RoboDK station: ex2.rdk

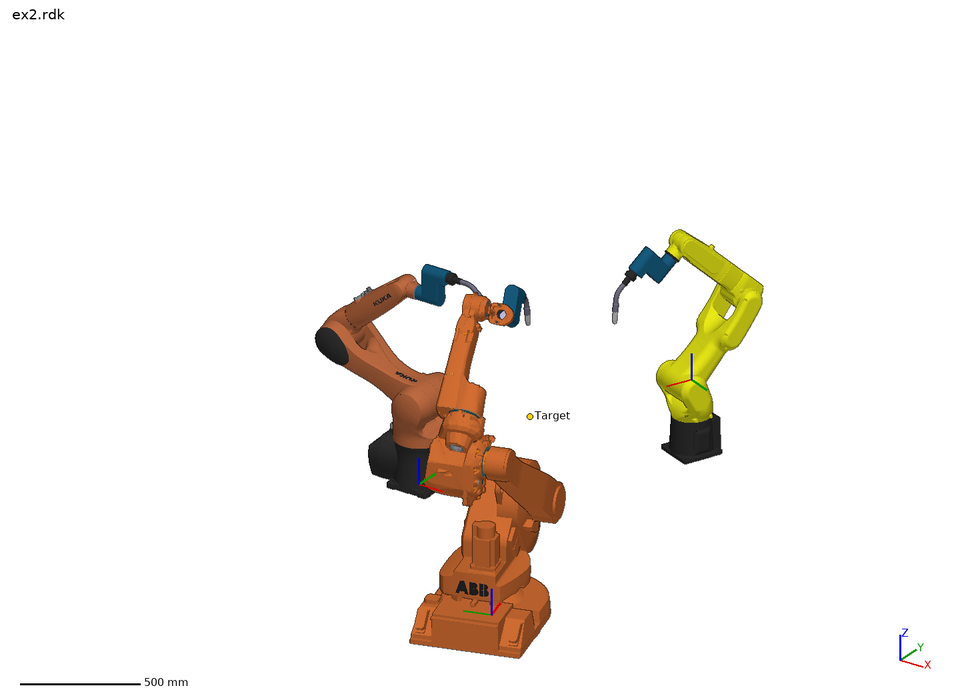
[picture v0: the station drawn from its stored meshes, robots at their saved joint values, targets as dots, program paths as lines]
Station ex2. Poses are relative to the parent item; angles as X-Y-Z fixed-axis rotations.
  - frame KUKA KR 6 R900 sixx Base at (0, 0, 0) mm
    - robot KUKA KR 6 R900 sixx: 6 axes, payload 6 kg, reach 901 mm, repeatability 0.03 mm, weight 52 kg
        modified DH rows (alpha deg, a mm, theta deg, d mm): 0, 0, 0, 400; -90, 25, 0, 0; 0, 455, -90, 0; -90, 35, 0, 420; 90, 0, 0, 0; -90, 0, 180, 80
        joint limits [-170, -190, -120, -185, -120, -350] to [170, 45, 156, 185, 120, 350]; home [0, -154.452, 115.025, 0, 39.427, 0]; saved at [0, -154.452, 115.025, 0, 39.427, 0]
      - tool Weld gun KUKA, TCP at (-4, 0, 371.3) mm, rotated rx 0 ry 45 rz 0 deg, size 299.9 x 60 x 318.3 mm
    - target Target (Cartesian target) at (564.87, 0, 471.83) mm, rotated rx -180 ry 0 rz -180 deg; joints [0, -116.511, 123.863, 0, 37.648, 0] of KUKA KR 6 R900 sixx
  - frame ABB IRB 1600ID-4/1.5 Base at (957.87, -842.99, 0) mm, rotated rx 0 ry 0 rz 107.3 deg
    - robot ABB IRB 1600ID-4/1.5: 6 axes, payload 4 kg, reach 1500 mm, repeatability 0.02 mm, weight 250 kg
        modified DH rows (alpha deg, a mm, theta deg, d mm): 0, 0, 0, 486.5; -90, 150, -90, 0; 0, 700, 0, 0; -90, 110, 0, 640; 90, 0, 0, 0; -90, 0, 180, 200
        joint limits [-180, -90, -238, -155, -90, -200] to [180, 150, 79, 155, 135, 200]; home [0, -52.548, 13.111, 0, 71.84, 0]; saved at [0, -52.548, 13.111, 0, 71.84, 0]
      - tool Weld gun ABB, TCP at (-4, 0, 371.3) mm, rotated rx 45 ry 0 rz 90 deg, size 299.9 x 60 x 318.3 mm
  - frame Fanuc LR Mate 200iD/7L Base at (872.61, 731.91, 437.52) mm, rotated rx 0 ry 0 rz -111.87 deg
    - robot Fanuc LR Mate 200iD/7L: 6 axes, payload 7 kg, reach 911 mm, repeatability 0.03 mm, weight 27 kg
        modified DH rows (alpha deg, a mm, theta deg, d mm): 0, 0, 0, 330; -90, 50, -90, 0; 0, 440, 0, 0; -90, 35, 0, 420; 90, 0, 0, 0; -90, 0, 0, 80
        base shift (0, 0, -330) mm
        joint limits [-170, -100, -67, -190, -115, -360] to [170, 145, 213, 190, 115, 360]; home [0, -40.966, 43.328, 0, -84.792, 180]; saved at [0, -40.966, 43.328, 0, -84.792, 180]
      - tool Weld gun Fanuc, TCP at (-4, 0, 371.3) mm, rotated rx -45 ry 0 rz -90 deg, size 299.9 x 60 x 318.3 mm
  - Python program DoWeld (listed below)
  - Python program DoWeldAll (listed below)

--- Python program DoWeld ---
from robolink import *    # API to communicate with RoboDK
from robodk import *      # basic matrix operations

# Any interaction with RoboDK must be done through
# Robolink()
RDK = Robolink()

# get the robot item:
robot = RDK.ItemUserPick('Select a robot for welding', ITEM_TYPE_ROBOT)
if not robot.Valid():
    raise Exception("Operation cancelled by user")

# get the home joints target
home = robot.JointsHome()

# get the reference welding target:
target = RDK.Item('Target')

# get the reference frame and set it to the robot
reference = target.Parent()
robot.setFrame(reference)

# get the pose of the target (4x4 matrix):
poseref = target.Pose()
pose_approach = poseref*transl(0,0,-100)

# move the robot to home, then to the center:
robot.MoveJ(home)
robot.MoveJ(pose_approach)
robot.MoveL(target)

# make an hexagon around the center:
for i in range(7):
    ang = i*2*pi/6 #angle: 0, 60, 120, ...
    posei = poseref*rotz(ang)*transl(200,0,0)*rotz(-ang)
    robot.MoveL(posei)

# move back to the center, then home:
robot.MoveL(target)
robot.MoveL(pose_approach)
robot.MoveJ(home)

--- Python program DoWeldAll ---
from robolink import *    # API to communicate with RoboDK
from robodk import *      # basic matrix operations
import threading
import queue

#----------------------------------------------
# Function definitions and global variable declarations

# Global variables used to synchronize the robot movements
# These variables are managed by SyncSet() and SynchWait()

SYNC_COUNT = 0
SYNC_TOTAL = 0
SYNC_ID = 0
lock = threading.Lock()

def SyncSet(total_sync):
    """SyncSet will set the number of total robot programs (threads) that must be synchronized togeter.
    Every time SyncSet is called SYNC_ID is increased by one."""
    global SYNC_COUNT
    global SYNC_TOTAL
    global SYNC_ID
    with lock:
        SYNC_COUNT = 0
        SYNC_TOTAL = total_sync
        SYNC_ID = SYNC_ID + 1
        #print('SyncSet')

def SyncWait():
    """SyncWait will block the robot movements for a robot when necessary, synchronizing the movements sequentially.
    Use SyncSet(nrobots) to define how many robots must be synchronized together."""
    global SYNC_COUNT
    # Save a local variable with the sync event id
    sync_id = SYNC_ID
    with lock:
        # Increase the number of threads that are synchronized
        SYNC_COUNT += 1

    # Move to the next sync event if all threads reached the SyncWait (SYNC_COUNT = SYNC_TOTAL)
    if SYNC_COUNT >= SYNC_TOTAL:
        SyncSet(SYNC_TOTAL)
        return

    # Wait for a SynchSet to move forward
    while sync_id >= SYNC_ID:
        time.sleep(0.0001)


# Main procedure to move each robot
def DoWeld(q, robotname):
    # Any interaction with RoboDK must be done through Robolink()
    # Each robot movement requires a new Robolink() object (new link of communication).
    # Two robots can't be moved by the same communication link.

    rdk = Robolink()

    # get the robot item:
    robot = rdk.Item(robotname)

    # get the home joints target
    home = robot.JointsHome()

    # get the reference welding target:
    target = rdk.Item('Target')

    # get the reference frame and set it to the robot
    reference = target.Parent()
    robot.setFrame(reference)

    # get the pose of the target (4x4 matrix):
    poseref = target.Pose()
    pose_approach = poseref*transl(0,0,-100)

    # move the robot to home, then to the center:
    robot.MoveJ(home)
    robot.MoveJ(pose_approach)
    SyncWait()
    robot.MoveL(target)

    # make an hexagon around the center:
    for i in range(7):
        ang = i*2*pi/6 #angle: 0, 60, 120, ...
        posei = poseref*rotz(ang)*transl(200,0,0)*rotz(-ang)
        SyncWait()
        robot.MoveL(posei)

    # move back to the center, then home:
    SyncWait()
    robot.MoveL(target)
    robot.MoveL(pose_approach)
    robot.MoveJ(home)
    q.put('Robot %s finished' % robotname)

#----------------------------------------
# Python program start

# retrieve all available robots in the RoboDK station (as a list of names)
RDK = Robolink()
robots = RDK.ItemList(ITEM_TYPE_ROBOT)
print(robots)

# retrieve the number of robots to synchronize together
nrobots = len(robots)
SyncSet(nrobots)

# the queue allows sharing messages between threads
q = queue.Queue()

# Start the DoWeld program for all robots. Each robot will run on a separate thread.
threads = []
for i in range(nrobots):
    robotname = robots[i]
    t = threading.Thread(target=DoWeld, args = (q, robotname))
    t.daemon = True
    t.start()
    threads.append(t)

# wait for every thead to finish
for x in threads:
    x.join()
    print(q.get())

print('Main program finished')
